FUNCTION_BLOCK LRealComparer EXTENDS Object IMPLEMENTS IComparer
VAR
	_ClassName : STRING := __POUNAME();
END_VAR

{attribute 'monitoring' := 'call'}
PROPERTY ClassName : STRING
GET
ClassName := _ClassName;
END_GET
END_PROPERTY

{attribute "object_name" := "Compare"}
METHOD Compare : COMPARISION_RESULT
VAR_INPUT
	left : __SYSTEM.AnyType;
	right : __SYSTEM.AnyType;
END_VAR
VAR
	leftPointer : POINTER TO LREAL; 
	rightPointer : POINTER TO LREAL; 
END_VAR
IF left.pValue = 0 AND right.pValue = 0 THEN
	Compare := COMPARISION_RESULT.FIRST_EQUAL_TO_SECOND;
	RETURN;
END_IF

IF left.pValue = 0 THEN
	Compare := COMPARISION_RESULT.FIRST_LESS_THAN_SECOND;
	RETURN;	
END_IF

IF right.pValue = 0 THEN
	Compare := COMPARISION_RESULT.FIRST_GREATER_THAN_SECOND;
	RETURN;	
END_IF

leftPointer := left.pValue;
rightPointer := right.pValue;

IF leftPointer^ < rightPointer^ THEN
	Compare := COMPARISION_RESULT.FIRST_LESS_THAN_SECOND;
ELSIF leftPointer^ > rightPointer^ THEN
	Compare := COMPARISION_RESULT.FIRST_GREATER_THAN_SECOND;
ELSE
	Compare := COMPARISION_RESULT.FIRST_EQUAL_TO_SECOND;	
END_IF
END_METHOD

{attribute 'monitoring' := 'call'}
PROPERTY Size : ULINT
GET
Size := XSIZEOF(THIS^);
END_GET
END_PROPERTY

END_FUNCTION_BLOCK

(* stored: Version 1.1.0.1
   POU LRealComparer: Id {f4e21534-0e97-4f45-9e9f-9fc5128a94f9}, SpecialFunc None
   Property ClassName: Id {c7b91571-bf88-48e0-bcfa-79b7189f7876}
   Get Get: Id {07b7f3e7-f1b8-4851-80cc-39e5356991ac}
   Method Compare: Id {4c67832f-1632-413f-a01f-80ee0feddaaa}
   Property Size: Id {d9d53921-7b08-48ef-888d-d76d25d2b4e7}
   Get Get: Id {c2f8c3a5-7acc-4512-ad96-cf0a19ce7b60} *)
